// TIA Portal V20 export
// export: Created 2025-12-01T14:57:20.7771103Z, ExportSetting None, DisplayName Totally Integrated Automation Portal, DisplayVersion V20 Update 3, DisplayName TIA Portal Openness, DisplayVersion V20 Update 3, DisplayName TIA Portal Version Control Interface, DisplayVersion V20 Update 3, DisplayName STEP 7 Professional, DisplayVersion V20 Update 3, DisplayName STEP 7 Safety, DisplayVersion V20 Update 2, DisplayName WinCC Basic/Comfort/Advanced, DisplayVersion V20 Update 3, DisplayName WinCC Professional, DisplayVersion V20 Update 3, DisplayName WinCC Unified, DisplayVersion V20 Update 3
DATA_BLOCK "DB2100_VarSeguridades"   // DB2100, F_DB
{ S7_Optimized_Access := 'TRUE' }
// stored: AutoNumber false
   VAR
      ALWAYS_ON_SEG : Bool;   // Always ON
      ALWAYS_OFF_SEG : Bool;   // Always OFF
      FP_1_seg : Bool;
      ACK_Next_01 : Bool;
      ACK_Next_02 : Bool;
      ACK_Next_03 : Bool;
      ACK_Next_04 : Bool;
      ACK_Next_05 : Bool;
      ACK_Next_06 : Bool;
      ACK_Next_07 : Bool;
      ACK_Next_08 : Bool;
      ACK_Next_09 : Bool;
      ACK_Next_10 : Bool;
      ACK_Next_11 : Bool;
      ACK_Next_12 : Bool;
      ACK_Next_13 : Bool;
      ACK_Next_14 : Bool;
      ACK_Next_15 : Bool;
      ACK_Next_16 : Bool;
      ACK_Next_17 : Bool;
      ACK_Next_18 : Bool;
      ACK_Next_19 : Bool;
      ACK_Next_20 : Bool;
      ACK_Next_21 : Bool;
      ACK_Next_22 : Bool;
      ACK_Next_23 : Bool;
      ACK_Next_24 : Bool;
      ACK_Next_25 : Bool;
      ACK_Next_26 : Bool;
      ACK_Next_27 : Bool;
      ACK_Next_28 : Bool;
      ACK_Next_29 : Bool;
      ACK_Next_30 : Bool;
      ACK_Next_31 : Bool;
      ACK_Next_32 : Bool;
      ACK_Next_33 : Bool;
      ACK_Next_34 : Bool;
      ACK_Next_35 : Bool;
      ACK_Next_36 : Bool;
      ACK_Next_37 : Bool;
      ACK_Next_38 : Bool;
      ACK_Next_39 : Bool;
      ACK_Next_40 : Bool;
      LP_Sinoptico_1 : Word;
      LP_Sinoptico_2 : Word;
      LP_Sinoptico_3 : Word;
      LP_Sinoptico_4 : Word;
      LP_Sinoptico_5 : Word;
      LP_Sinoptico_6 : Word;
      LP_Sinoptico_7 : Word;
      LP_Sinoptico_8 : Word;
      LP_Sinoptico_9 : Word;
      LP_Sinoptico_10 : Word;
      LP_Sinoptico_11 : Word;
      LP_Sinoptico_12 : Word;
      LP_Sinoptico_13 : Word;
      LP_Sinoptico_14 : Word;
      LP_Sinoptico_15 : Word;
      LP_Sinoptico_16 : Word;
      LP_Sinoptico_17 : Word;
      LP_Sinoptico_18 : Word;
      LP_Sinoptico_19 : Word;
      LP_Sinoptico_20 : Word;
      LP_Sinoptico_21 : Word;
      LP_Sinoptico_22 : Word;
      LP_Sinoptico_23 : Word;
      LP_Sinoptico_24 : Word;
      LP_Sinoptico_25 : Word;
      LP_Sinoptico_26 : Word;
      LP_Sinoptico_27 : Word;
      LP_Sinoptico_28 : Word;
      LP_Sinoptico_29 : Word;
      LP_Sinoptico_30 : Word;
      BS_Sinoptico_1 : Word;
      BS_Sinoptico_2 : Word;
      BS_Sinoptico_3 : Word;
      BS_Sinoptico_4 : Word;
      BS_Sinoptico_5 : Word;
      BS_Sinoptico_6 : Word;
      BS_Sinoptico_7 : Word;
      BS_Sinoptico_8 : Word;
      BS_Sinoptico_9 : Word;
      BS_Sinoptico_10 : Word;
      BS_Sinoptico_11 : Word;
      BS_Sinoptico_12 : Word;
      BS_Sinoptico_13 : Word;
      BS_Sinoptico_14 : Word;
      BS_Sinoptico_15 : Word;
      BS_Sinoptico_16 : Word;
      BS_Sinoptico_17 : Word;
      BS_Sinoptico_18 : Word;
      BS_Sinoptico_19 : Word;
      BS_Sinoptico_20 : Word;
      BS_Sinoptico_21 : Word;
      BS_Sinoptico_22 : Word;
      BS_Sinoptico_23 : Word;
      BS_Sinoptico_24 : Word;
      BS_Sinoptico_25 : Word;
      BS_Sinoptico_26 : Word;
      BS_Sinoptico_27 : Word;
      BS_Sinoptico_28 : Word;
      BS_Sinoptico_29 : Word;
      BS_Sinoptico_30 : Word;
      BS_Sinoptico_31 : Word;
      BS_Sinoptico_32 : Word;
      BS_Sinoptico_33 : Word;
      BS_Sinoptico_34 : Word;
      BS_Sinoptico_35 : Word;
      BS_Sinoptico_36 : Word;
      BS_Sinoptico_37 : Word;
      BS_Sinoptico_38 : Word;
      BS_Sinoptico_39 : Word;
      BS_Sinoptico_40 : Word;
      BS_Sinoptico_41 : Word;
      BS_Sinoptico_42 : Word;
      BS_Sinoptico_43 : Word;
      BS_Sinoptico_44 : Word;
      BS_Sinoptico_45 : Word;
      BS_Sinoptico_46 : Word;
      BS_Sinoptico_47 : Word;
      BS_Sinoptico_48 : Word;
      BS_Sinoptico_49 : Word;
      BS_Sinoptico_50 : Word;
   END_VAR
BEGIN
END_DATA_BLOCK
